// Common discoverable base interface for registered entities.
INTERFACE I_Generic EXTENDS __SYSTEM.IQueryInterface, I_Debug

END_INTERFACE

(* stored: Version 1.1.0.1
   Itf I_Generic: Id {b8d5ed71-9568-4c56-ba31-ef1af9c39847} *)
